// TwinCAT 3 PLC project Plc
// Title: InvokeCSharp
// Company: Inxton
// Author: Inxton-Dev-Team
// ProjectVersion: 0.0.0.0
// ProgramVersion: 3.1.4023.0
// libraries:
//   Tc2_Standard, * (Beckhoff Automation GmbH)
//   Tc2_System, * (Beckhoff Automation GmbH)
//   Tc3_Module, * (Beckhoff Automation GmbH)
//   TcoCore, 0.5.0.829 (Vortex.Library)
//   TcoData, 0.5.0.829 (Vortex.Library)
// project tree:
//   / PlcTask.TcTTO
//   POUs/ App.TcPOU, Data.TcDUT, DataManager.TcPOU, MAIN.TcPOU, Person.TcDUT
// real-time tasks:
//   TASK PlcTask: cycle T#10ms, priority 20, ADS port 350

CONFIGURATION Plc
    RESOURCE PLC ON TwinCAT3
        TASK PlcTask(INTERVAL := T#10ms, PRIORITY := 20);
        PROGRAM MAIN WITH PlcTask : MAIN;
    END_RESOURCE
END_CONFIGURATION

// ---- POUs/Data.TcDUT
TYPE Data EXTENDS TcoData.TcoEntity :
STRUCT
	DataId : STRING;
    Person_0 :Person;
    Person_1 :Person;
    Person_2 :Person;
    Person_3 :Person;
    Person_4 :Person;
    Person_5 :Person;
    Person_6 :Person;
    Person_7 :Person;
    Person_8 :Person;
    Person_9 :Person;
END_STRUCT
END_TYPE

// ---- POUs/Person.TcDUT
TYPE Person :
STRUCT
	FirstName : STRING;
	LastName : STRING;
	Age : INT;
	Birthday : DATE;
	BirthTown : STRING;
END_STRUCT
END_TYPE

// ---- POUs/MAIN.TcPOU
PROGRAM MAIN
VAR
	App : App;
END_VAR

App.Run();

END_PROGRAM

// ---- POUs/App.TcPOU
FUNCTION_BLOCK App EXTENDS TcoCore.TcoContext
VAR
	Step: INT;
	GenerateDataTask: TcoCore.TcoRemoteTask(THIS^);
	DataManager : DataManager(THIS^);
END_VAR

(*~
	<docu>
		<summary>
			Main method of the TcoContext. This is the entry point of any control logic that belongs to this context. 
			The call of this method is ensured by calling the <c>InstanceName.Run()</c> method, and it must not be called explicitly.
			This method is abstract, and it must be overridden in derived block.
		</summary>
	</docu>
~*)
METHOD PROTECTED  Main
VAR
	ID : STRING;
END_VAR
GenerateDataTask();
DataManager();

CASE Step OF
	0 : 
		IF GenerateDataTask.Invoke().Done THEN
			Step := Step + 10;
		END_IF
	10 :
		Step:= Step + 10;
	20 :
		ID := ULINT_TO_STRING(THIS^._rtc.TickClock());
		IF DataManager.Create(ID).Done THEN
			Step := 0;
		END_IF
END_CASE
END_METHOD

END_FUNCTION_BLOCK

// ---- POUs/DataManager.TcPOU
FUNCTION_BLOCK DataManager EXTENDS TcoData.TcoDataExchange
VAR
	_data : Data;
END_VAR

SUPER^();

END_FUNCTION_BLOCK
